SYSTEM VisualTest (* System Configuration *)
  (* Standard: 61499-1 *)
  (* Version 0.3, 2003-12-05, JHC, Rockwell Automation, Renamed from NEWSYSTEM. *)
  (* Version 0.2, 2002-11-05, JHC, Rockwell Automation, Fixed missing (empty) FBD in Application. *)
  (* Version 0.1, 2002-01-17, JHC, Rockwell Automation, Minor cleanup *)
  (* Version 0.0, 2000-05-27, JHC, Rockwell Automation *)
  APPLICATION APP1
  END_APPLICATION
  DEVICE DISPLAY : ImageDev(Length := 300, Height := 300)
    RESOURCE resource : ImageResource
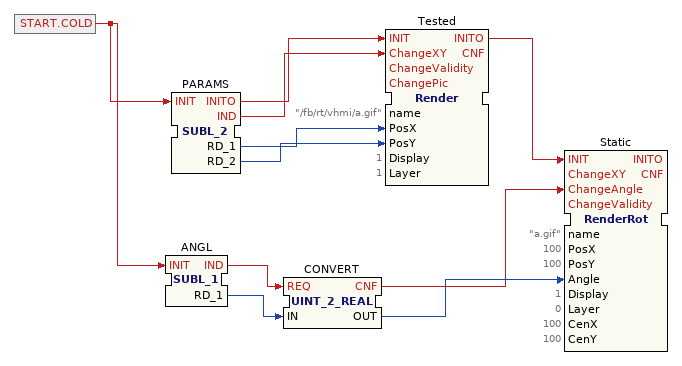
      FBS
        PARAMS : SUBL_2;
        ANGL : SUBL_1;
        Tested : Render(name := "/fb/rt/vhmi/a.gif", Display := 1, Layer := 1);
        CONVERT : UINT_2_REAL;
        Static : RenderRot(name := "a.gif", PosX := 100, PosY := 100, Layer := 0, Display := 1, CenX := 100, CenY := 100);
      END_FBS
      EVENT_CONNECTIONS
        START.COLD TO PARAMS.INIT;
        START.COLD TO ANGL.INIT;
        PARAMS.INITO TO Tested.INIT;
        PARAMS.IND TO Tested.ChangeXY;
        ANGL.IND TO CONVERT.REQ;
        Tested.INITO TO Static.INIT;
        CONVERT.CNF TO Static.ChangeAngle;
      END_CONNECTIONS
      DATA_CONNECTIONS
        PARAMS.RD_1 TO Tested.PosX;
        ANGL.RD_1 TO CONVERT.IN;
        PARAMS.RD_2 TO Tested.PosY;
        CONVERT.OUT TO Static.Angle;
      END_CONNECTIONS
    END_RESOURCE
  END_DEVICE
  DEVICE HMI : FRAME_DEVICE(BOUNDS := [0,301,300,100], GRID := [1,1])
    RESOURCE RES1 : PANEL_RESOURCE
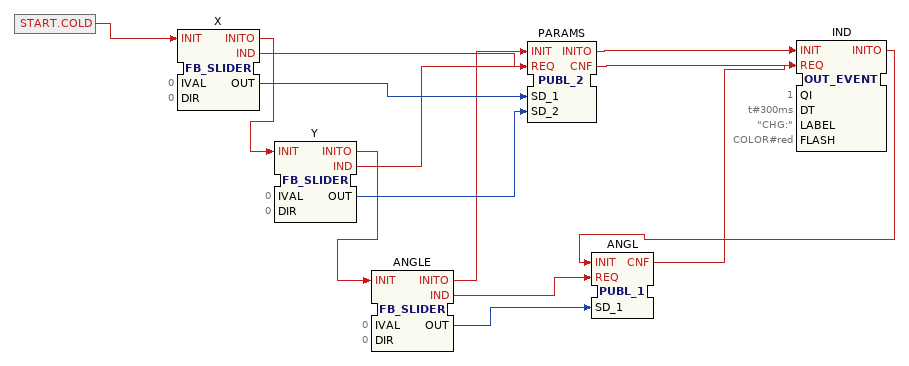
      FBS
        X : FB_SLIDER(IVAL := 0, DIR := 0);
        Y : FB_SLIDER(IVAL := 0, DIR := 0);
        PARAMS : PUBL_2;
        ANGLE : FB_SLIDER(IVAL := 0, DIR := 0);
        IND : OUT_EVENT(QI := 1, DT := t#300ms, LABEL := "CHG:", FLASH := COLOR#red);
        ANGL : PUBL_1;
      END_FBS
      EVENT_CONNECTIONS
        START.COLD TO X.INIT;
        X.INITO TO Y.INIT;
        ANGLE.INITO TO PARAMS.INIT;
        Y.INITO TO ANGLE.INIT;
        Y.IND TO PARAMS.REQ;
        X.IND TO PARAMS.REQ;
        PARAMS.INITO TO IND.INIT;
        PARAMS.CNF TO IND.REQ;
        IND.INITO TO ANGL.INIT;
        ANGLE.IND TO ANGL.REQ;
        ANGL.CNF TO IND.REQ;
      END_CONNECTIONS
      DATA_CONNECTIONS
        X.OUT TO PARAMS.SD_1;
        Y.OUT TO PARAMS.SD_2;
        ANGLE.OUT TO ANGL.SD_1;
      END_CONNECTIONS
    END_RESOURCE
  END_DEVICE
END_SYSTEM
